{attribute 'qualified_only'}
{attribute 'strict'}
TYPE E_GrundfosMagna3ControlMode :
(
	constantSpeed := 0,
	constantTemperature_Heating := 1,
	constantTemperature_Cooling := 2,
	temperatureDifference := 3,
	pressureDifference := 4,
	proportionalPressureControl :=5
);
END_TYPE

(* stored: Version 1.1.0.1, ProductVersion 3.1.4024.10
   DUT E_GrundfosMagna3ControlMode: Id {0ebc95ca-56b0-475f-9f3e-553d6515e4b2} *)
